// TwinCAT 3 PLC project TCPIP_Client
// ProgramVersion: 3.1.4024.0
// libraries:
//   Tc2_Standard, * (Beckhoff Automation GmbH)
//   Tc2_System, * (Beckhoff Automation GmbH)
//   Tc2_TcpIp, * (Beckhoff Automation GmbH)
//   Tc2_Utilities, * (Beckhoff Automation GmbH)
//   Tc3_Module, * (Beckhoff Automation GmbH)
// project tree:
//   DUTs/ E_ConnectionSteps.TcDUT (not stored)
//   GVLs/ GVL.TcGVL
//   / PlcTask.TcTTO (not stored)
//   POUs/ FB_Client.TcPOU, FB_ClientConnection.TcPOU (not stored), MAIN.TcPOU
//   POUs/Helper POUs/ FB_FrameFifo.TcPOU (not stored), FB_LogFifo.TcPOU
// real-time tasks:
//   TASK PlcTask: cycle T#10ms, priority 20, ADS port 350

// ---- GVLs/GVL.TcGVL
{attribute 'qualified_only'}
VAR_GLOBAL CONSTANT
	PLCPRJ_BUFFER_SIZE						: UDINT := 1000;	(* Max. internal fifo/receiver buffer size *)

	PLCPRJ_CLIENT_SEND_CYCLE_TIME			: TIME := T#1S;
	PLCPRJ_RECEIVE_POLLING_TIME				: TIME := T#100MS;
	PLCPRJ_RECEIVE_TIMEOUT					: TIME := T#600S;

	(* Some project specific error codes *)
	PLCPRJ_ERROR_RECEIVE_TIMEOUT			: UDINT := 16#8101;	(* Receive timeout *)
	PLCPRJ_ERROR_SENDFIFO_OVERFLOW			: UDINT := 16#8102;	(* Send fifo overflow *)
	PLCPRJ_ERROR_RECFIFO_OVERFLOW			: UDINT := 16#8103;	(* Receive fifo overflow *)
END_VAR

VAR_GLOBAL
END_VAR

// ---- POUs/FB_Client.TcPOU
FUNCTION_BLOCK FB_Client
VAR_INPUT
	sSrvNetID	: T_AmsNetID	:= '';				(* TwinCAT TCP/IP server network address *)
	sRemoteHost	: T_IPv4Addr 	:= '127.0.0.1';		(* Server network address *)
	nRemotePort	: UDINT 		:= 200;				(* Server port number *)
	bEnable		: BOOL 			:= FALSE;			(* TRUE => enable client data exchange, FALSE => disable *)
	bLog		: BOOL 			:= FALSE;			(* TRUE => Enable log message output, FALSE => Disable *)
	sPrefix		: STRING 		:= 'CLIENT::';		(* Log message description string (allows the identification of log message source) *)
	fbTx 						: FB_FrameFifo;		(* Tx fifo *)
	fbRx 						: FB_FrameFifo;		(* Rx fifo *)
END_VAR
VAR_OUTPUT
	bConnected	: BOOL 			:= FALSE;			(* TCP/IP connection state *)
	RxText		: String[255];
END_VAR
VAR
	fbConnection	: FB_ClientConnection;			(* Client connection/data exchange control function block *)
	fbLog			: FB_LogFifo;					(* Log/debug/error fifo *)
END_VAR

(*-------------------------- Trigger data exchange -----------------------------------------------*)
fbConnection( 	sSrvNetID := sSrvNetID, fbTx := fbTx, fbRx := fbRx, fbLog := fbLog, 
				bEnable := bEnable, sRemoteHost := sRemoteHost, nRemotePort := nRemotePort,  
				bLog := bLog, sPrefix := sPrefix, bConnected=>bConnected, RxText => RxText );

END_FUNCTION_BLOCK

// ---- POUs/Helper POUs/FB_LogFifo.TcPOU
(* Log/debug/error message fifo *)
FUNCTION_BLOCK FB_LogFifo
VAR_INPUT
	bLog		: BOOL 		:= FALSE;(* TRUE => Enable log message output, FALSE => Disable *)
	sPrefix		: STRING 	:= 'Unknown::';(* Log message description string (allows the identification of log message source) *)
	
	sMessage	: STRING 	:= '';(* String message to add (write) to the fifo *)
	nErrID		: UDINT 	:= 0;(* Error code to add (write) to the fifo *)
	hSocket		: T_HSOCKET;(* Socket connection handle *)
END_VAR
VAR_OUTPUT
	bOk			: BOOL;(* TRUE = New entry added or removed succesfully, FALSE = Fifo overflow or fifo empty *)
	sGet		: T_MaxString := '';(* String entry removed (read) from fifo *)
	nCount		: UDINT := 0;(* Number of fifo entries *)
END_VAR
VAR
	fbBuffer 	: FB_StringRingBuffer;(* Basic (lower level) string buffer control function block *)
	buffer		: ARRAY[0..GVL.PLCPRJ_BUFFER_SIZE] OF BYTE;(* Internal buffer memory *)
	sSource		: T_MaxString;	
	sPut		: T_MaxString;
END_VAR

;

ACTION Clear:
(* Clears all fifo entries *)
fbBuffer.A_Reset( 	pBuffer := ADR( buffer ), cbBuffer := SIZEOF( buffer ), 
					bOk=>bOk, nCount=>nCount, getValue=>sGet );
END_ACTION

ACTION Error:
(* Adds new fifo entry *)
IF nErrID = 0 THEN
	sSource := '::Error: 0x';
ELSIF ( nErrID AND 16#80000000) = 16#80000000 THEN
	IF nErrID = 16#80072746 THEN
		sSource := '::Win32 error (the connection is reset by remote side): 0x';
	ELSE
		sSource := '::Win32 error: 0x';
	END_IF
ELSIF (nErrID AND 16#00008100) = 16#00008100 THEN
	CASE nErrID OF
		GVL.PLCPRJ_ERROR_RECEIVE_TIMEOUT:
			sSource := '::PLC sample project receive timeout error: 0x';
		GVL.PLCPRJ_ERROR_SENDFIFO_OVERFLOW:
			sSource := '::PLC sample project send fifo overflow error: 0x';
		GVL.PLCPRJ_ERROR_RECFIFO_OVERFLOW:
			sSource := '::PLC sample project receive fifo overflow error: 0x';
	ELSE
		sSource := '::Other PLC sample project error: 0x';
	END_CASE
ELSIF (nErrID AND 16#00008000) = 16#00008000 THEN
	sSource := '::Internal TCP/IP Connection Server error: 0x';
ELSE
	sSource := '::TwinCAT System error: 0x';
END_IF

sPut := CONCAT( CONCAT( CONCAT( sPrefix, sMessage ), sSource ), DWORD_TO_HEXSTR( nErrID AND 16#FFFF, 0, FALSE ) ); 

fbBuffer.A_AddTail( pBuffer:= ADR(buffer), cbBuffer:= SIZEOF(buffer),
					putValue:= sPut, bOk=>bOk, nCount=>nCount );
IF bOk THEN
	IF bLog THEN(* Log error message *)
		ADSLOGSTR( ADSLOG_MSGTYPE_ERROR OR ADSLOG_MSGTYPE_LOG, '%s', sPut );	
	END_IF
END_IF
END_ACTION

ACTION Message:
(* Adds new fifo entry *)
sPut := CONCAT( CONCAT( sPrefix, sMessage ), CONCAT( '::', HSOCKET_TO_STRING(hSocket) ) );
fbBuffer.A_AddTail( pBuffer:= ADR(buffer), cbBuffer:= SIZEOF(buffer),
					putValue:= sPut, bOk=>bOk, nCount=>nCount );
IF bOk THEN
	IF bLog THEN(* Log information message *)
		ADSLOGSTR( ADSLOG_MSGTYPE_HINT OR ADSLOG_MSGTYPE_LOG, '%s', sPut );	
	END_IF
END_IF
END_ACTION

ACTION Remove:
(* Removes oldest fifo entry *)
IF nCount = 0 THEN
	sGet := '';
	bOk := FALSE;
	RETURN;
END_IF

fbBuffer.A_RemoveHead( pBuffer:= ADR(buffer), cbBuffer:= SIZEOF(buffer),
						getValue=>sGet, bOk=>bOk, nCount=>nCount );
END_ACTION

END_FUNCTION_BLOCK

// ---- POUs/MAIN.TcPOU
PROGRAM MAIN
VAR
		
	sSrvNetID		: T_AmsNetID	:= '';
	bScannerEnable	: BOOL 			:= TRUE;
	bLaserEnable	: BOOL 			:= TRUE;
	bLog			: BOOL			:= FALSE;
	fbClient_ABC 	: FB_Client 	:= ( sRemoteHost := '127.0.0.1',
										 nRemotePort := 8500,
										 sPrefix := '' );
										
	fbCloseAll		: FB_SocketCloseAll;
	bInitialize		: BOOL := TRUE;
	bConnected		: BOOL;
	nErrId			: UDINT;
	data_send_flag  : BOOL;
	Msg			: STRING := '';
	Send_msg		: STRING := '';
	Received_msg	: STRING := '';
END_VAR


	fbCloseAll( sSrvNetID := sSrvNetID, bExecute:= bInitialize );
	IF fbCloseAll.bBusy OR fbCloseAll.bError THEN
		nErrId := fbCloseAll.nErrId;
		RETURN;
	END_IF
	
	bInitialize := FALSE;
	fbClient_ABC	( sSrvNetId := sSrvNetID, bEnable := bScannerEnable	, bLog := bLog, bConnected => bConnected );
	
	IF data_send_flag THEN
		Send_msg := CONCAT(Msg, '$R');
		fbClient_ABC.fbTx.AddTail( sPut := Send_msg); //$R = Carriage Return [CR]
		data_send_flag := false;
	END_IF
	
	Received_msg := fbClient_ABC.RxText;

END_PROGRAM
